// TIA Portal V17 export
// export: Created 2022-02-03T14:45:11.3239726Z, ExportSetting WithDefaults, DisplayName Totally Integrated Automation Portal, DisplayVersion V17, DisplayName TIA Portal Openness, DisplayVersion V17, DisplayName TIA Portal Version Control Interface, DisplayVersion V17, DisplayName SINAMICS Startdrive Advanced, DisplayVersion V17, DisplayName SINAMICS Startdrive G130, G150, S120, S150, SINAMICS MV, S210, DisplayVersion V17, DisplayName SINAMICS Startdrive G110M, G120, G120C, G120D, G120P, G115D, DisplayVersion V17, DisplayName STEP 7 Professional, DisplayVersion V17, DisplayName STEP 7 Safety, DisplayVersion V17, DisplayName WinCC Advanced, DisplayVersion V17
FUNCTION "Signal" : Void   // FC2, LAD
VERSION : 0.1
// stored: Access Published, AutoNumber true, IsIECCheckEnabled false, SetENOAutomatically false, UDAEnableTagReadback false
   VAR_INPUT
      operation : Bool;
      conveyorIn : "typeConveyorInput";
      occupiedBay : Array[#FIRSTBAY..#LASTBAY] of Bool;
      conveyorFault : Bool;
      weightOk : Bool;
      currentStoreFull : Bool;
   END_VAR
   VAR_OUTPUT
      operationModeLED : Bool;
      conveyorFaultLED : Bool;
      restartManualLED : Bool;
      restartAutoLED : Bool;
      weightFaultLED : Bool;
      messageBits : Word;
   END_VAR
   VAR_IN_OUT
      conveyorOUT : "typeConveyorOutput";
      restartMan : Bool;
      restartAuto : Bool;
      instLGF_Frequency : "LGF_Frequency";
   END_VAR
   VAR_TEMP
      tempFrequ2Hz : Bool;
   END_VAR
   VAR CONSTANT
      FIRSTBAY : UInt := 1;
      LASTBAY : UInt := 3;
   END_VAR
BEGIN

REGION Network 1
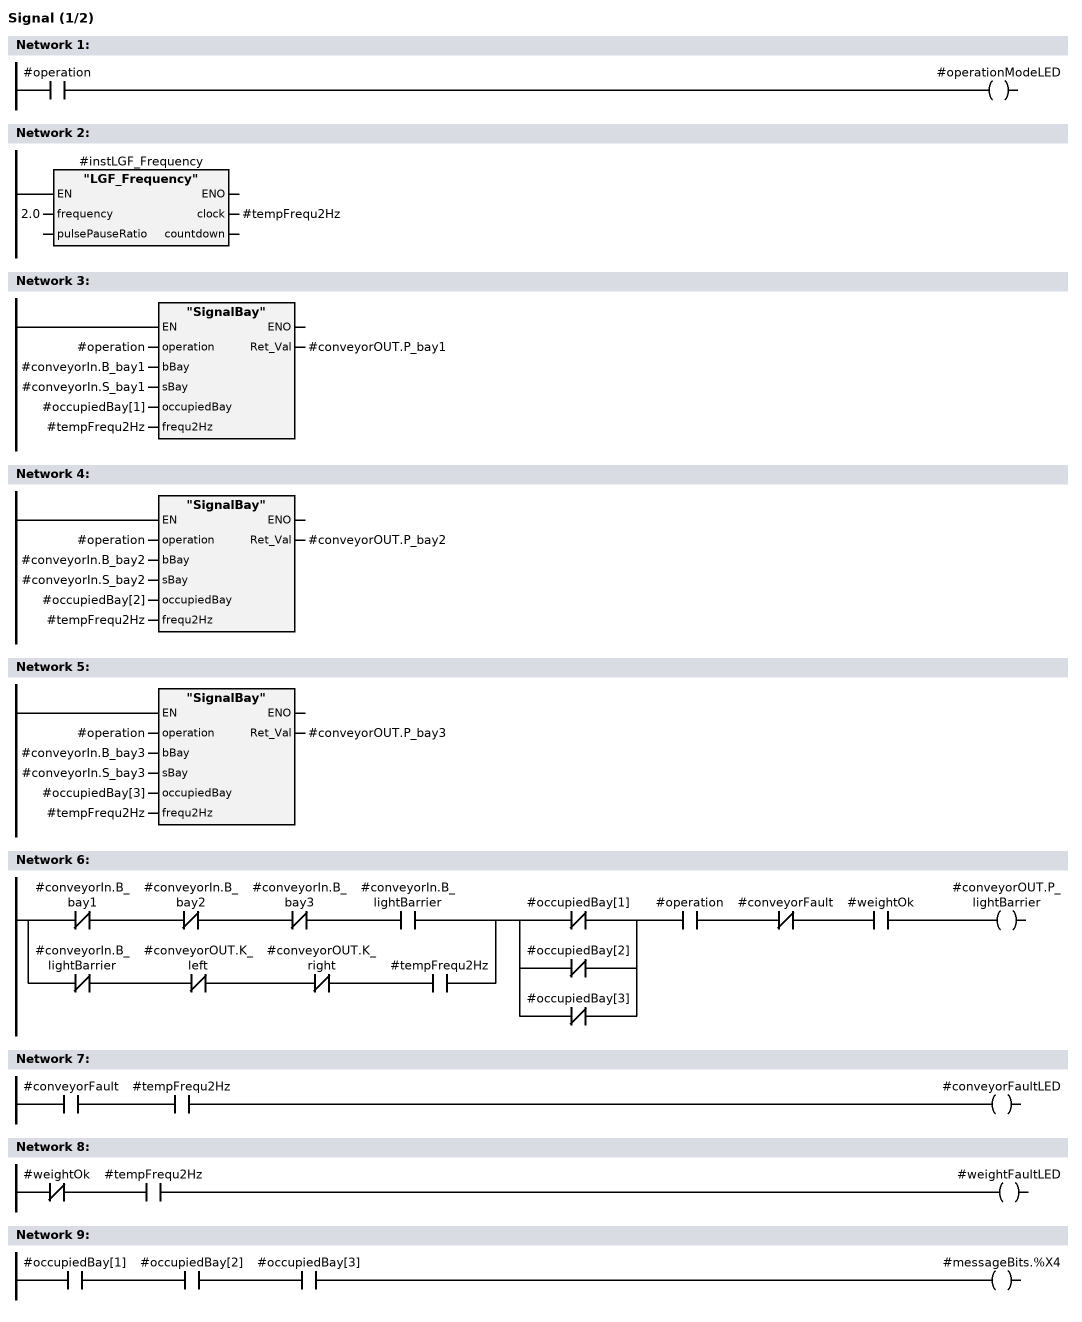
   RUNG wire#powerrail
      Contact( #operation )
      Coil( #operationModeLED )
   END_RUNG
   // the same network as SCL:
   #operationModeLED := #operation;
END_REGION

REGION Network 2
   RUNG wire#powerrail
      #instLGF_Frequency(frequency := 2.0, pulsePauseRatio :=, clock => #tempFrequ2Hz, countdown =>)
   END_RUNG
   // the same network as SCL:
   #instLGF_Frequency(frequency := 2.0, clock => #tempFrequ2Hz);   // "LGF_Frequency"
END_REGION

REGION Network 3
   RUNG wire#powerrail
      "SignalBay"(operation := #operation, bBay := #conveyorIn.B_bay1, sBay := #conveyorIn.S_bay1, occupiedBay := #occupiedBay[1], frequ2Hz := #tempFrequ2Hz, Ret_Val => #conveyorOUT.P_bay1)
   END_RUNG
   // the same network as SCL:
   #conveyorOUT.P_bay1 := "SignalBay"(operation := #operation,
                           bBay := #conveyorIn.B_bay1,
                           sBay := #conveyorIn.S_bay1,
                           occupiedBay := #occupiedBay[1],
                           frequ2Hz := #tempFrequ2Hz);
END_REGION

REGION Network 4
   RUNG wire#powerrail
      "SignalBay"(operation := #operation, bBay := #conveyorIn.B_bay2, sBay := #conveyorIn.S_bay2, occupiedBay := #occupiedBay[2], frequ2Hz := #tempFrequ2Hz, Ret_Val => #conveyorOUT.P_bay2)
   END_RUNG
   // the same network as SCL:
   #conveyorOUT.P_bay2 := "SignalBay"(operation := #operation,
                           bBay := #conveyorIn.B_bay2,
                           sBay := #conveyorIn.S_bay2,
                           occupiedBay := #occupiedBay[2],
                           frequ2Hz := #tempFrequ2Hz);
END_REGION

REGION Network 5
   RUNG wire#powerrail
      "SignalBay"(operation := #operation, bBay := #conveyorIn.B_bay3, sBay := #conveyorIn.S_bay3, occupiedBay := #occupiedBay[3], frequ2Hz := #tempFrequ2Hz, Ret_Val => #conveyorOUT.P_bay3)
   END_RUNG
   // the same network as SCL:
   #conveyorOUT.P_bay3 := "SignalBay"(operation := #operation,
                           bBay := #conveyorIn.B_bay3,
                           sBay := #conveyorIn.S_bay3,
                           occupiedBay := #occupiedBay[3],
                           frequ2Hz := #tempFrequ2Hz);
END_REGION

REGION Network 6
   RUNG wire#powerrail
      I_Contact( #conveyorIn.B_bay1 )
      I_Contact( #conveyorIn.B_bay2 )
      I_Contact( #conveyorIn.B_bay3 )
      Contact( #conveyorIn.B_lightBarrier )
      wire#w1
      I_Contact( #occupiedBay[1] )
      wire#w2
      Contact( #operation )
      I_Contact( #conveyorFault )
      Contact( #weightOk )
      Coil( #conveyorOUT.P_lightBarrier )
   END_RUNG
   RUNG wire#powerrail
      I_Contact( #conveyorIn.B_lightBarrier )
      I_Contact( #conveyorOUT.K_left )
      I_Contact( #conveyorOUT.K_right )
      Contact( #tempFrequ2Hz )
   END_RUNG wire#w1
   RUNG wire#w1
      I_Contact( #occupiedBay[2] )
   END_RUNG wire#w2
   RUNG wire#w1
      I_Contact( #occupiedBay[3] )
   END_RUNG wire#w2
   // the same network as SCL:
   #conveyorOUT.P_lightBarrier := ((NOT #conveyorIn.B_bay1 AND NOT #conveyorIn.B_bay2 AND NOT #conveyorIn.B_bay3 AND #conveyorIn.B_lightBarrier) OR (NOT #conveyorIn.B_lightBarrier AND NOT #conveyorOUT.K_left AND NOT #conveyorOUT.K_right AND #tempFrequ2Hz)) AND (NOT #occupiedBay[1] OR NOT #occupiedBay[2] OR NOT #occupiedBay[3]) AND #operation AND NOT #conveyorFault AND #weightOk;
END_REGION

REGION Network 7
   RUNG wire#powerrail
      Contact( #conveyorFault )
      Contact( #tempFrequ2Hz )
      Coil( #conveyorFaultLED )
   END_RUNG
   // the same network as SCL:
   #conveyorFaultLED := #conveyorFault AND #tempFrequ2Hz;
END_REGION

REGION Network 8
   RUNG wire#powerrail
      I_Contact( #weightOk )
      Contact( #tempFrequ2Hz )
      Coil( #weightFaultLED )
   END_RUNG
   // the same network as SCL:
   #weightFaultLED := NOT #weightOk AND #tempFrequ2Hz;
END_REGION

REGION Network 9
   RUNG wire#powerrail
      Contact( #occupiedBay[1] )
      Contact( #occupiedBay[2] )
      Contact( #occupiedBay[3] )
      Coil( #messageBits.%X4 )
   END_RUNG
   // the same network as SCL:
   #messageBits.%X4 := #occupiedBay[1] AND #occupiedBay[2] AND #occupiedBay[3];
END_REGION

REGION Network 10
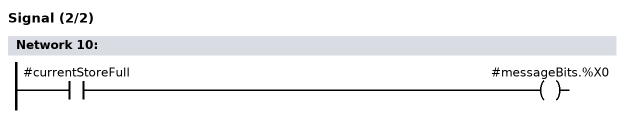
   RUNG wire#powerrail
      Contact( #currentStoreFull )
      Coil( #messageBits.%X0 )
   END_RUNG
   // the same network as SCL:
   #messageBits.%X0 := #currentStoreFull;
END_REGION
END_FUNCTION
